TYPE ST_SafetyStatus :
STRUCT
    bSafeToRun : BOOL;
    bEStopActive : BOOL;
    bSafetyRelayOK : BOOL;
    bRelayDiscrepancy : BOOL;
    bGuardDoorOpen : BOOL;
    bSTOActive : BOOL;
    bDriveInhibit : BOOL;
    bNetworkHealthy : BOOL;
    bWatchdogHealthy : BOOL;
    bDriveReadyHealthy : BOOL;
    bAnyLimitTripped : BOOL;
    abLimitPosActive : ARRAY[1..2] OF BOOL;
    abLimitNegActive : ARRAY[1..2] OF BOOL;
    nSafetyStatusWord : UINT;
END_STRUCT
END_TYPE

(* stored: Version 1.1.0.1
   DUT ST_SafetyStatus: Id {E889E37D-0E06-5844-53DD-B57AF12A3DB3} *)
